FUNCTION_BLOCK PushToStartLogic
VAR_INPUT
	StartEquipment:BOOL;
END_VAR
VAR_OUTPUT
	RelayCommandToStart:BOOL;
	RelayCommandToStop:BOOL;
END_VAR
VAR
     StartTrig:R_Trig;
	 Stoptrig:F_Trig;
	
	 StartCounter:INT;
	 StopCounter:INT;	
END_VAR

///Logic for the push button

///Start logic 
StartTrig(CLK:=StartEquipment,q=>);

IF StartTrig.Q THEN
   RelayCommandToStart:=TRUE;
END_IF

IF RelayCommandToStart THEN
   StartCounter:=StartCounter+1;
IF StartCounter=50 THEN
   RelayCommandToSTart:=FALSE;	
   StartCounter:=0;
END_IF
END_IF
   
 ///Stop logic
 StopTrig(CLK:=StartEquipmenT,Q=>);
 IF StopTrig.Q THEN
	RelayCommandToStop:=TRUE;
 END_IF
 
 IF RelayCommandToStop THEN
	StopCounter:=StopCounter+1;
    IF StopCounter=50 THEN
	   RelayCommandToStop:=FALSE;
	   StopCounter:=0;
    END_IF
 END_IF

END_FUNCTION_BLOCK

(* stored: Version 1.1.0.1, ProductVersion 3.1.4024.0
   POU PushToStartLogic: Id {44988478-a266-4239-8cc6-41d513efc741}, SpecialFunc None *)
